// TIA Portal V18 export
TYPE "UDT_vAO"
// stored: IsFailsafeCompliant false
   STRUCT
      rInput : Real;   // Value for AO
      cMOA : Byte := 0;   // Mode Manual/Off/Auto
      cFuncSystemID : Byte := 0;
      cFuncVar : Byte := 0;
      cMemory : Byte := 0;
      rManOutput : Real;   // Manual output
      iOutput : Int;   // Output for DAC
   END_STRUCT;
END_TYPE
